TEXTLIST tlVacuumStep_V2
  0 = 'Init'
  1 = 'Wait for obtaining atmospheric pressure'
  5 = 'Setup new test'
  10 = 'Waiting for ext test premission '
  15 = 'Stating new cycle'
  20 = 'Waiting for end of cycle'
  25 = 'Waiting for pressure low value'
  30 = 'Waiting for doors open'
  90 = 'Error obtained'
  91 = 'Waiting for reset'
  95 = 'Reset confirmed'
  50 = 'Manual mode'
   = ''
END_TEXTLIST

(* stored: Version 1.1.0.1, ProductVersion 3.1.4024.13
   TextList tlVacuumStep_V2: Id {7add8e82-6746-4c77-baeb-4180d12d69b3} *)
